// TIA Portal V20 export
DATA_BLOCK "LPFE_PRTBuffer"   // DB246
TITLE = Buffer of RequestOrderInfo messages
// Buffer to store record messages (7,8) until distributed
// stored: Access Published, MemoryReserve 100, Namespace PFE
   VAR
      buffer { ExternalAccessible := 'False'; ExternalVisible := 'False'; ExternalWritable := 'False'} : Array[0.._.LE_NUMBER_MESSAGES_PRT_BUFFER] of "LPFE_typePFEDataReqEnvelope";   // Buffer where record messages are taken from
      mgmtBuffer { ExternalAccessible := 'False'; ExternalVisible := 'False'; ExternalWritable := 'False'} : "LPFE_typeMsgBuffer";   // Mgmt Structure of buffer where record messages are taken from
   END_VAR
BEGIN
END_DATA_BLOCK
